Staubli VAL3: save_AxisType.pjx

Parameters version=s7.2.1 stackSize=5000 millimeterUnit=true
Data file=save_AxisType.dtx
Library alias=io path=Disk://io/io.pjx
